TYPE "FeedMachine_TXT"
VERSION : 0.1
// Block: FeedMachine_TXT
   STRUCT
      par_Group : String;
      Desc_P01_Man_Vel_BWD : String;
      Desc_P02_Man_Vel_FWD_High : String;
      Desc_P03_Man_Vel_FWD_Low : String;
      Um_P01 : String;
      Um_P02 : String;
      Um_P03 : String;
   END_STRUCT;

END_TYPE
